// TIA Portal V21 export
TYPE "LBC_typeDiagnostics"
TITLE = LBC_typeDiagnostic
// Module related diagnostic information
   STRUCT
      status { ExternalWritable := 'False'} : Word;   // 16#0000-16#7FFF: Status of the FB 16#8000-16#FFFF: Error identification
      subfunctionStatus { ExternalWritable := 'False'} : Word;   // Status or return value of called FB's, FCs, system blocks or other status information
      stateNumber { ExternalWritable := 'False'} : DInt;   // State in the state machine of the block where the error occurred
   END_STRUCT;
END_TYPE
